Universal Robots PolyScope program: eventcounter-advance.urp

ProgramRoot directory=/home/ur/ursim-3.1/programs/Support site/EventCounter; kinematics=(a=[0, -0.425, -0.39225, 0, 0, 0], d=[0.08916, 0, 0, 0.10915, 0.09465, 0.0823], alpha=[1.5708, 0, 0, 1.5708, -1.5708, 0], deltaTheta=[0, 0, 0, 0, 0, 0], status=notInitialized); lastSavedInVersion=(project__name=Polyscope, major__version=3, minor__version=1, svn__revision=18024, build__date=Jul 07 2015, 15:18:49); name=eventcounter-advance; programVersion=(project__name=Polyscope, major__version=3, minor__version=1, svn__revision=17195, build__date=Mar 11 2015, 13:02:28); robotEnvironmentFileName=default; serialNumberRobot=2015350001
  InitVariables 
  MainProgram cartesianAcceleration=1.2; cartesianSpeed=0.25; jointAcceleration=1.3962634015954636; jointSpeed=1.0471975511965976; sharedProcessMoveBlendRadius=0.025; motionType=JOINT_SPACE
    Wait 
    Assignment expr=ExpressionIONode; operatorValueType=INTEGER; valueSource=EXPRESSION; variable=False
    If expr=ExpressionVariableNode and  not  False ≟ False; type=IF_NODE
      Assignment expr=ExpressionVariableNode+1; operatorValueType=INTEGER; valueSource=EXPRESSION; variable=0
      If expr=ExpressionVariableNode≥24; type=IF_NODE
        Assignment expr=0; operatorValueType=INTEGER; valueSource=EXPRESSION; variable=0
        Assignment expr=True; operatorValueType=INTEGER; valueSource=EXPRESSION; variable=False
    Assignment expr=ExpressionVariableNode; operatorValueType=INTEGER; valueSource=EXPRESSION; variable=False
    If expr=ExpressionVariableNode≟ True; type=IF_NODE
      Move cartesianAcceleration=1.2; cartesianSpeed=0.25; jointAcceleration=1.3962634015954636; jointSpeed=1.0471975511965976; sharedProcessMoveBlendRadius=0.025; motionType=JOINT_SPACE
        Waypoint blendRadius=0.05; cartesianAcceleration=1.2; cartesianSpeed=0.25; jointAcceleration=1.3962634015954636; jointSpeed=1.0471975511965976; nextMotionTime=2.0; stoppoint=true; useSharedBlendParameter=true; useSharedParameters=true; position=TCP in base x=-120.113 y=-431.763 z=146.073 mm, rx=-0.0012 ry=3.1163 rz=0.0389 rad; joints [-91.713, -98.956, -126.223, -46.295, 91.393, -1.776] deg; positionType=FIXED_POSITION; waypointPoseInFeatureCoordinates=(pos=(x=-0.12011317028458361, y=-0.4317631667637431, z=0.14607252291477704), rot=(x=-0.0012209830284081382, y=3.1162764812408743, z=0.03889191616813277)); name=Waypoint_1
        Waypoint blendRadius=0.05; cartesianAcceleration=1.2; cartesianSpeed=0.25; jointAcceleration=1.3962634015954636; jointSpeed=1.0471975511965976; nextMotionTime=2.0; stoppoint=true; useSharedBlendParameter=true; useSharedParameters=true; position=TCP in base x=-2.927 y=-448.15 z=146.073 mm, rx=-0.4131 ry=3.0923 rz=0.0438 rad; joints [-76.541, -98.956, -126.223, -46.295, 91.393, -1.776] deg; positionType=FIXED_POSITION; waypointPoseInFeatureCoordinates=(pos=(x=-0.002927142710124496, y=-0.4481495706627684, z=0.14607252291477704), rot=(x=-0.41305782136505986, y=3.0922610949710903, z=0.04375804659402105)); name=Waypoint_2
      Assignment expr=False; operatorValueType=INTEGER; valueSource=EXPRESSION; variable=False
